// TIA Portal V20 export
TYPE "UDT_Service_StepOrderRawDataMedium"
   STRUCT
      stepOrder : Array[0..199] of "UDT_Service_StepOrder";
      parameterIndex : Array[0..511] of Byte;
   END_STRUCT;
END_TYPE
